// TIA Portal V19 export
TYPE "lexchangetray_typeUnEmn_signalTM_Simulation"
// Type: Bool
// stored: Access Published
   STRUCT
      w : Bool;
   END_STRUCT;
END_TYPE
